(* IEC 61131-3 sources: AXOpen/src/components.drives/app/src/Sandbox, 1 file *)

(* ---- SandboxContext.st ---- *)
NAMESPACE AXOpen.Components.Drives
    {S7.extern=ReadWrite}
    CLASS SandboxContext EXTENDS AXOpen.Core.AxoContext
        VAR PUBLIC
            _manualControl : BOOL;
            PlcInputs : ARRAY [0..10] OF BYTE;
            PlcOutputs : ARRAY [0..10] OF BYTE;
            _rootObject :   AxoObject;
            _testDrive  : AXOpen.Components.Drives.AxoDriveExample;
        END_VAR

        METHOD PROTECTED OVERRIDE Main
            THIS.InitializeRootObject(_rootObject);
            IF(_manualControl) THEN
                _testDrive.ActivateManualControl();
            END_IF;
            _testDrive.Run(parent           :=  _rootObject,
                            refAxisIn       :=  REF(PlcInputs),
                            refAxisOut      :=  REF(PlcOutputs),
                            Enable          :=  TRUE,
                            EnablePositive  :=  TRUE,
                            EnableNegative  :=  TRUE);
        END_METHOD
    END_CLASS
END_NAMESPACE
